INTERFACE I_FlagList EXTENDS Debug.I_Debug

METHOD Cap : UDINT
VAR_INPUT
END_VAR
END_METHOD

METHOD GetByPos : Results.Result
VAR_INPUT
	nPos			: UDINT;
END_VAR
VAR_OUTPUT
	iFlag			: I_Flag;
END_VAR
END_METHOD

METHOD GetByTag : Results.Result
VAR_INPUT
	iTag			: Tags.I_Tag;
END_VAR
VAR_OUTPUT
	iFlag			: I_Flag;
	nPos			: UDINT;
END_VAR
END_METHOD

METHOD GetExtender : FlagListExtender
VAR_INPUT
END_VAR
END_METHOD

METHOD IsReleased : BOOL
VAR_INPUT
END_VAR
END_METHOD

METHOD Length : UDINT
VAR_INPUT
END_VAR
END_METHOD

METHOD Release : FlagListExtender;
END_METHOD

END_INTERFACE

(* stored: Version 1.1.0.1
   Itf I_FlagList: Id {3c2f77c0-ccec-4d42-845e-c4c167ab7784}
   Folder Get: Id {ed8ad8a0-4d12-4472-a44c-4d9d7c31f2ce}
   Folder Other: Id {310d51f6-f6ef-4d14-96c8-9a2189e22f49}
   Method Cap: Id {d89b32cf-fa65-4ca3-b7e3-11d076ac49e0}
   Method GetByPos: Id {80681568-58cb-48b5-8808-9a7f271ec616}
   Method GetByTag: Id {79ef193c-92d1-4a81-87f9-d0209112765d}
   Method GetExtender: Id {c17953b4-d32c-471a-a346-1f0eefe9989d}
   Method IsReleased: Id {85b025d0-ba0a-43d4-8d7b-eeaac6420119}
   Method Length: Id {6b41d57f-cfb9-42ef-91d7-9731c0971080}
   Method Release: Id {5cf4ed2c-8714-43f8-afb0-bfd8624c3e0e} *)
